{attribute 'GeneratedUsingTerminal: AES-D-BC-ECAT Gen2-0001'}
{attribute addProperty BoxType "AES-D-BC-ECAT Gen2-0001"}
{attribute addProperty Id "digital_Data_IAT %I*ARRAY[0..31] OF USINT32"}
{attribute addProperty CRC "1374483313"}
{attribute addProperty Size "32"}
TYPE Inputs_23559BB0 EXTENDS TcoIo.InputBase_8311D824 :
STRUCT
	{attribute addProperty Name "digital_Data_I"}
	digital_Data_I AT %I* : ARRAY[0..31] OF USINT;
END_STRUCT
END_TYPE

(* stored: Version 1.2.0.0, ProductVersion 3.1.4024.9
   DUT Inputs_23559BB0: Id {602a507e-7d8e-03a0-3a98-d65ba1c0f005} *)
